TYPE ST_Heightlimit :
STRUCT
	LOW:   INT;
	HIGH:  INT;
	
END_STRUCT
END_TYPE

(* stored: Version 1.1.0.1, ProductVersion 3.1.4024.13
   DUT ST_Heightlimit: Id {0a40893a-a1af-4cdb-af9d-50f041b8a80e} *)
